// TIA Portal V19 export
FUNCTION_BLOCK "Infeed"   // FB41, LAD
TITLE = Sinamics Infeed / SINAMICS INFEED CONTROL WITH TELEGRAM 370 1/1 Word
// stored: Access Published, MemoryReserve 100, SetENOAutomatically false
   VAR_INPUT
      EStopDly : Bool;   // Emergency Stop delay (1=OK)
      Rst : Bool;   // Reset alarms
      Enable : Bool;   // Enable infeed (cmd Start)
      Tel370_HWID : HW_IO;   // Telegram 370 for SinaInfeed
      AccessPoint : HW_IO;   // AccesPoint for SinaParaS
      AxisID : USInt;   // Axis ID for SinaParaS
      TokenChain : Int;   // Number of token chain for SinaParaS
      Simulation : Bool;
      Delay_PowerOff { ExternalAccessible := 'False'; ExternalVisible := 'False'; ExternalWritable := 'False'} : Time := T#5M;
   END_VAR
   VAR_OUTPUT
      Ready : Bool;   // Infeed ready
      Running : Bool;   // Infeed running (Enabled)
      AlarmPresence : Bool;   // Cumulative alarm presence
      WarningPresence : Bool;   // Cumulative warning presence
   END_VAR
   VAR_IN_OUT
      Alarm : "InfeedAlr";
      Warning : "InfeedWng";
      Diag : "TO_Diagnostic";
   END_VAR
   VAR
      ReadAlarm : "RW_SINAMICS_Par";
      ReadWarning : "RW_SINAMICS_Par";
      SinaInfeed : SinaInfeed;
      ComunicationON : Bool;
      EnableInfeed : Bool;
      tonComunicationON : IEC_TIMER;
      tonPowered : IEC_TIMER;
      tonTimeoutActivation : IEC_TIMER;
      tonPowerOff : IEC_TIMER;
   END_VAR
BEGIN

REGION Network 1 (SCL): Info
   //=============================================================================
   //PM FORMING
   //-----------------------------------------------------------------------------
   // Library: StandardBlocks
   // Tested with: S7-1518TF
   // Engineering: TIA Portal V18
   // Restrictions: -
   // Requirements: S7-1500
   // Functionality: Sinamics Infeed device
   //
   // v1.0.0  28/12/2022 
   // v1.1.0  14/02/2022 Simulation added
   //=============================================================================
   //
END_REGION

REGION Network 2: Comunication ON
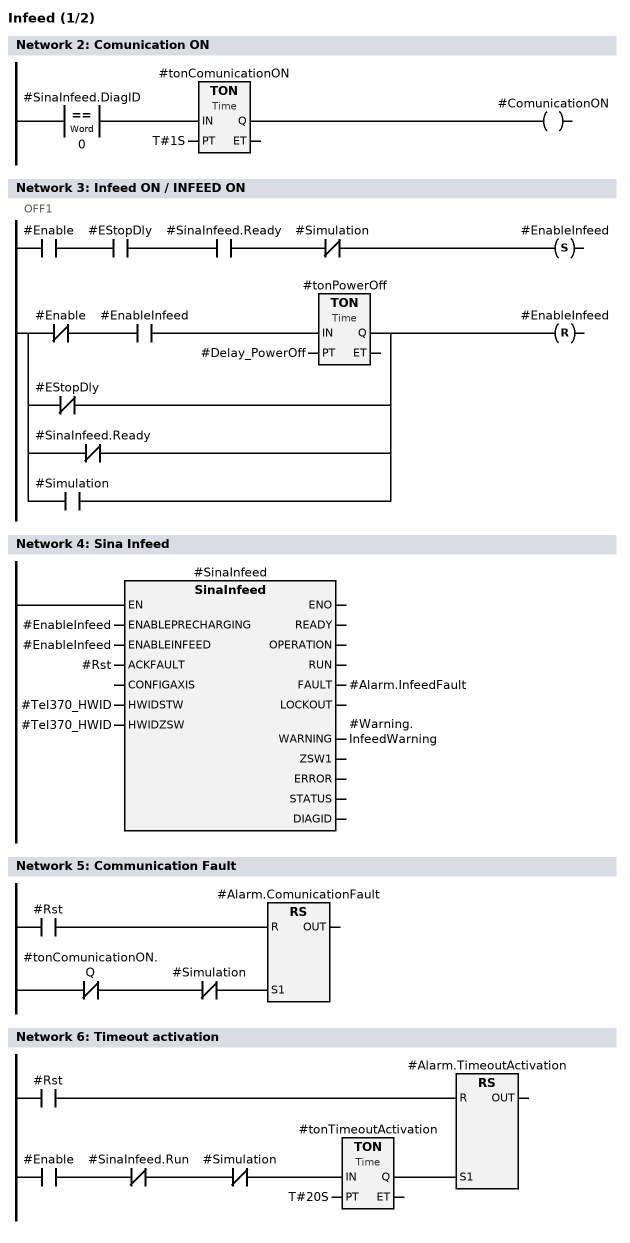
   RUNG wire#powerrail
      { S7_Templates := "SrcType := Word" } EQ_Contact(in1 := #SinaInfeed.DiagID, in2 := 0)
      { S7_Templates := "time_type := Time" } #tonComunicationON.TON(pt := T#1S, et =>)
      Coil( #ComunicationON )
   END_RUNG
   // the same network as SCL:
   #tonComunicationON.TON(IN := #SinaInfeed.DiagID = 0, PT := T#1S);
   #ComunicationON := #tonComunicationON.Q;
END_REGION

REGION Network 3: Infeed ON / INFEED ON
   // OFF1
   RUNG wire#powerrail
      Contact( #Enable )
      Contact( #EStopDly )
      Contact( #SinaInfeed.Ready )
      I_Contact( #Simulation )
      S_Coil( #EnableInfeed )
   END_RUNG
   RUNG wire#powerrail
      I_Contact( #Enable )
      Contact( #EnableInfeed )
      { S7_Templates := "time_type := Time" } #tonPowerOff.TON(pt := #Delay_PowerOff, et =>)
      wire#w1
      R_Coil( #EnableInfeed )
   END_RUNG
   RUNG wire#powerrail
      I_Contact( #EStopDly )
   END_RUNG wire#w1
   RUNG wire#powerrail
      I_Contact( #SinaInfeed.Ready )
   END_RUNG wire#w1
   RUNG wire#powerrail
      Contact( #Simulation )
   END_RUNG wire#w1
   // the same network as SCL:
   IF #Enable AND #EStopDly AND #SinaInfeed.Ready AND NOT #Simulation THEN #EnableInfeed := TRUE; END_IF;
   #tonPowerOff.TON(IN := NOT #Enable AND #EnableInfeed, PT := #Delay_PowerOff);
   IF #tonPowerOff.Q OR NOT #EStopDly OR NOT #SinaInfeed.Ready OR #Simulation THEN
       #EnableInfeed := FALSE;
   END_IF;
END_REGION

REGION Network 4: Sina Infeed
   RUNG wire#powerrail
      #SinaInfeed.SinaInfeed(EnablePrecharging := #EnableInfeed, EnableInfeed := #EnableInfeed, AckFault := #Rst, ConfigAxis :=, HWIDSTW := #Tel370_HWID, HWIDZSW := #Tel370_HWID, Ready =>, Operation =>, Run =>, Fault => #Alarm.InfeedFault, Lockout =>, Warning => #Warning.InfeedWarning, ZSW1 =>, Error =>, Status =>, DiagID =>)
   END_RUNG
   // the same network as SCL:
   #SinaInfeed(EnablePrecharging := #EnableInfeed,   // SinaInfeed
               EnableInfeed := #EnableInfeed,
               AckFault := #Rst,
               HWIDSTW := #Tel370_HWID,
               HWIDZSW := #Tel370_HWID,
               Fault => #Alarm.InfeedFault,
               Warning => #Warning.InfeedWarning);
END_REGION

REGION Network 5: Communication Fault
   RUNG wire#powerrail
      Contact( #Rst )
      S_RS(operand := #Alarm.ComunicationFault, s1 := wire#w1)
   END_RUNG
   RUNG wire#powerrail
      I_Contact( #tonComunicationON.Q )
      I_Contact( #Simulation )
   END_RUNG wire#w1
   // the same network as SCL:
   IF #Rst THEN
       #Alarm.ComunicationFault := FALSE;   // RS flip-flop
   END_IF;
   IF NOT #tonComunicationON.Q AND NOT #Simulation THEN #Alarm.ComunicationFault := TRUE; END_IF;
END_REGION

REGION Network 6: Timeout activation
   RUNG wire#powerrail
      Contact( #Rst )
      S_RS(operand := #Alarm.TimeoutActivation, s1 := wire#w1)
   END_RUNG
   RUNG wire#powerrail
      Contact( #Enable )
      I_Contact( #SinaInfeed.Run )
      I_Contact( #Simulation )
      { S7_Templates := "time_type := Time" } #tonTimeoutActivation.TON(pt := T#20S, et =>)
   END_RUNG wire#w1
   // the same network as SCL:
   #tonTimeoutActivation.TON(IN := #Enable AND NOT #SinaInfeed.Run AND NOT #Simulation, PT := T#20S);
   IF #Rst THEN
       #Alarm.TimeoutActivation := FALSE;   // RS flip-flop
   END_IF;
   IF #tonTimeoutActivation.Q THEN #Alarm.TimeoutActivation := TRUE; END_IF;
END_REGION

REGION Network 7: General Error
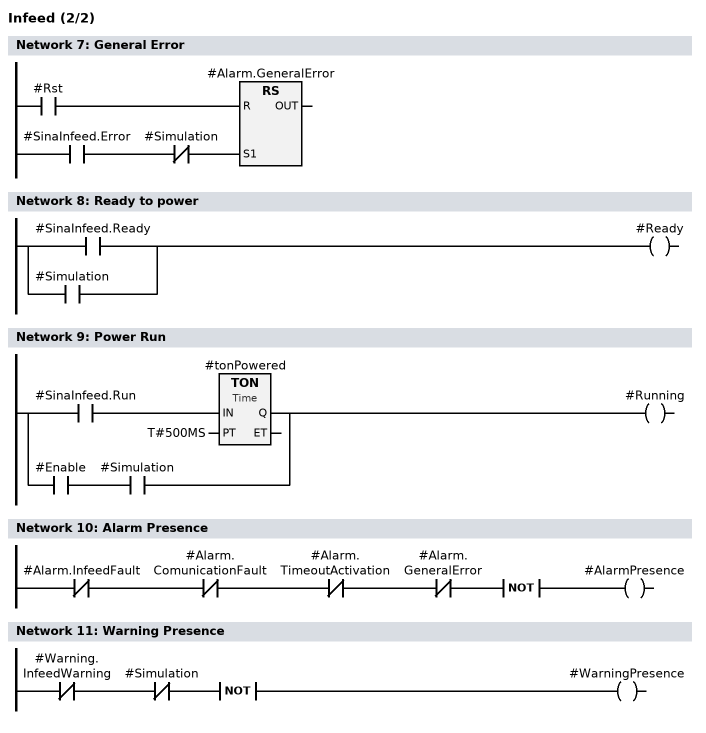
   RUNG wire#powerrail
      Contact( #Rst )
      S_RS(operand := #Alarm.GeneralError, s1 := wire#w1)
   END_RUNG
   RUNG wire#powerrail
      Contact( #SinaInfeed.Error )
      I_Contact( #Simulation )
   END_RUNG wire#w1
   // the same network as SCL:
   IF #Rst THEN
       #Alarm.GeneralError := FALSE;   // RS flip-flop
   END_IF;
   IF #SinaInfeed.Error AND NOT #Simulation THEN #Alarm.GeneralError := TRUE; END_IF;
END_REGION

REGION Network 8: Ready to power
   RUNG wire#powerrail
      Contact( #SinaInfeed.Ready )
      wire#w1
      Coil( #Ready )
   END_RUNG
   RUNG wire#powerrail
      Contact( #Simulation )
   END_RUNG wire#w1
   // the same network as SCL:
   #Ready := #SinaInfeed.Ready OR #Simulation;
END_REGION

REGION Network 9: Power Run
   RUNG wire#powerrail
      Contact( #SinaInfeed.Run )
      { S7_Templates := "time_type := Time" } #tonPowered.TON(pt := T#500MS, et =>)
      wire#w1
      Coil( #Running )
   END_RUNG
   RUNG wire#powerrail
      Contact( #Enable )
      Contact( #Simulation )
   END_RUNG wire#w1
   // the same network as SCL:
   #tonPowered.TON(IN := #SinaInfeed.Run, PT := T#500MS);
   #Running := #tonPowered.Q OR (#Enable AND #Simulation);
END_REGION

REGION Network 10: Alarm Presence
   RUNG wire#powerrail
      I_Contact( #Alarm.InfeedFault )
      I_Contact( #Alarm.ComunicationFault )
      I_Contact( #Alarm.TimeoutActivation )
      I_Contact( #Alarm.GeneralError )
      Not()
      Coil( #AlarmPresence )
   END_RUNG
   // the same network as SCL:
   #AlarmPresence := NOT (NOT #Alarm.InfeedFault AND NOT #Alarm.ComunicationFault AND NOT #Alarm.TimeoutActivation AND NOT #Alarm.GeneralError);
END_REGION

REGION Network 11: Warning Presence
   RUNG wire#powerrail
      I_Contact( #Warning.InfeedWarning )
      I_Contact( #Simulation )
      Not()
      Coil( #WarningPresence )
   END_RUNG
   // the same network as SCL:
   #WarningPresence := NOT (NOT #Warning.InfeedWarning AND NOT #Simulation);
END_REGION

REGION Network 12 (SCL): Diganostic

   #Diag.DeviceType := 2;
   #Diag.TO_SimulationActive := #Simulation;

   IF #AccessPoint > 0 AND #TokenChain > 0 AND NOT #Simulation THEN

       #ReadAlarm(Enable := #SinaInfeed.Fault,
                  ReadWrite := 0,
                  ParNo := 2131,
                  Index := 0,
                  AxisNo := #AxisID,
                  HW_ID := #AccessPoint,
                  TokenChain := #TokenChain);

       #ReadWarning(Enable := #SinaInfeed.Warning AND NOT #SinaInfeed.Fault,
                    ReadWrite := 0,
                    ParNo := 2132,
                    Index := 0,
                    AxisNo := #AxisID,
                    HW_ID := #AccessPoint,
                    TokenChain := #TokenChain);


       IF #SinaInfeed.Fault THEN
           IF #ReadAlarm.Done THEN
               #Diag.Drive_Message := REAL_TO_UINT(#ReadAlarm.ValueReadReal);
           END_IF;
       ELSIF #SinaInfeed.Warning THEN
           IF #ReadWarning.Done THEN
               #Diag.Drive_Message := REAL_TO_UINT(#ReadWarning.ValueReadReal);
           END_IF;
       ELSE
           #Diag.Drive_Message := 0;
       END_IF;

       #Diag.Drive_ErrorPresence := #SinaInfeed.Fault;
   ELSE
       #Diag.Drive_Message := 0;
       #Diag.Drive_ErrorPresence := FALSE;
   END_IF;

   IF #AlarmPresence THEN
       #Diag.MessageType := 2;
   ELSIF #WarningPresence THEN
       #Diag.MessageType := 1;
   ELSE
       #Diag.MessageType := 0;
   END_IF;
END_REGION
END_FUNCTION_BLOCK
